// TIA Portal project "canopen-snap7-interface" (V19)
// Using a S7-1200 PLC with the CM CANopen module to interact with a CANopen and Profinet network.

(* hardware
DEVICE "S7-1200 station_1"  S7-1200 Station
   slot 0: "Rack_0"  S7-1200 Rack  Rack  V1.0
   slot 1: "PLC_1"  CPU 1215C DC/DC/DC  6ES7 215-1AG40-0XB0  V4.6
   slot 101: "CM CANopen_1"  021620-B  V1.0
*)

// ===== PLC "PLC_1"  CPU 1215C DC/DC/DC =====

VAR_GLOBAL   // PLC tag table "Standard-Variablentabelle"
   "canOpenInputs" AT %I0.0 : "typeCanProcessImageInputs";
   "canOpenOutputs" AT %Q0.0 : "typeCanProcessImageOutputs";
   "Tag_1" AT %M110.0 : Bool;
   "Tag_2" AT %M110.1 : Bool;
END_VAR

VAR_GLOBAL CONSTANT   // PLC tag table "Standard-Variablentabelle"
   "Keiner" : Pip := 65535;
   "Automatische Aktualisierung" : Pip := 0;
   "TPA 1" : Pip := 1;
   "TPA 2" : Pip := 2;
   "TPA 3" : Pip := 3;
   "TPA 4" : Pip := 4;
   "TPA OB Servo" : Pip := 32768;
   "Local~HSC_1(1)" : Hw_Hsc := 257;
   "Local~HSC_2(1)" : Hw_Hsc := 258;
   "Local~HSC_3(1)" : Hw_Hsc := 259;
   "Local~HSC_4(1)" : Hw_Hsc := 260;
   "Local~HSC_5(1)" : Hw_Hsc := 261;
   "Local~HSC_6(1)" : Hw_Hsc := 262;
   "Local~AI_2_1" : Hw_SubModule := 263;
   "Local~DI_14_DQ_10_1(1)" : Hw_SubModule := 264;
   "Local~Pulse_1(1)" : Hw_Pwm := 265;
   "Local~Pulse_2(1)" : Hw_Pwm := 266;
   "Local~Pulse_3(1)" : Hw_Pwm := 267;
   "Local~Pulse_4(1)" : Hw_Pwm := 268;
   "Local~CM_CANopen_1(1)" : Port := 270;
   "OB_Main(1)" : OB_PCYCLE := 1;
   "Local~MC(1)" : Hw_SubModule := 51;
   "Local~Common(1)" : Hw_SubModule := 50;
   "Local~Device(1)" : Hw_Device := 32;
   "Local~Configuration(1)" : Hw_SubModule := 33;
   "Local~Exec(1)" : Hw_SubModule := 52;
   "Local(1)" : Hw_SubModule := 49;
   "Local~PROFINET-Schnittstelle_1" : Hw_Interface := 64;
   "Local~PROFINET-Schnittstelle_1~Port_1" : Hw_Interface := 65;
END_VAR

TYPE "typeCanProcessImageInputs"
VERSION : 0.1
   STRUCT
      BufferA : Struct
         SlaveDigitalInput1 : Byte;
         SlaveDigitalInput2 : Byte;
         SlaveAnalogInput1 : Int;
         SlaveAnalogInput2 : Int;
         SlaveAnalogInput3 : Int;
         SlaveAnalogInput4 : Int;
      END_STRUCT;
      BufferB : Struct
         SlaveDigitalInput1 : Byte;
         SlaveDigitalInput2 : Byte;
         SlaveAnalogInput1 : Int;
         SlaveAnalogInput2 : Int;
         SlaveAnalogInput3 : Int;
         SlaveAnalogInput4 : Int;
      END_STRUCT;
      ActiveBuffer : Byte;   // 0 = BufferA, 1 = BufferB. ActiveBuffer is the buffer the PC reads from, and the inactive buffer is the buffer the PLC updates from the input CAN process image.
   END_STRUCT;
END_TYPE

TYPE "typeCanProcessImageOutputs"
VERSION : 0.1
   STRUCT
      BufferA : Struct
         SlaveDigitalOutput1 : Byte;
         SlaveDigitalOutput2 : Byte;
         SlaveAnalogOutput1 : Int;
         SlaveAnalogOutput2 : Int;
         SlaveAnalogOutput3 : Int;
         SlaveAnalogOutput4 : Int;
         RequestID : UInt;
      END_STRUCT;
      BufferB : Struct
         SlaveDigitalOutput1 : Byte;
         SlaveDigitalOutput2 : Byte;
         SlaveAnalogOutput1 : Int;
         SlaveAnalogOutput2 : Int;
         SlaveAnalogOutput3 : Int;
         SlaveAnalogOutput4 : Int;
         RequestID : UInt;
      END_STRUCT;
      ResponseID : UInt;
      ActiveBuffer : Byte;   // 0 = BufferA, 1 = BufferB. ActiveBuffer is the buffer the PLC uses to write the output process image, and the inactive buffer is the buffer the PC writes to.
   END_STRUCT;
END_TYPE

DATA_BLOCK "MappedCanProcessImageOutputs"   // DB1
{ S7_Optimized_Access := 'FALSE' }
VERSION : 0.1
   VAR
      statCanProcessImageOutputs : "typeCanProcessImageOutputs";
   END_VAR
BEGIN
   statCanProcessImageOutputs.ActiveBuffer := 16#0;
END_DATA_BLOCK

DATA_BLOCK "ControlDB"   // DB3
{ S7_Optimized_Access := 'TRUE' }
VERSION : 0.1
   VAR
      CanProcessImageIn : Array[0..31] of Byte;
      CanProcessImageOut : Array[0..9] of Byte;
      ReadCanProcessImageBusy : Bool;
      ReadCanProcessImageError : Bool;
      ReadCanProcessImageSize : UInt;
      ReadCanProcessImageStatus : DWord;
      ReadCanProcessImageValid : Bool;
      WriteCanProcessImageBusy : Bool;
      WriteCanProcessImageError : Bool;
      WriteCanProcessImageSize : UInt;
      WriteCanProcessImageStatus : DWord;
      WriteCanProcessImageDone : Bool;
      ErrorRegisterReq : Bool;
      ErrorRegisterNode : Int;
      ErrorRegisterBusy : Bool;
      ErrorRegisterGenericError : Bool;
      ErrorRegisterCurrentError : Bool;
      ErrorRegisterVoltageError : Bool;
      ErrorRegisterTemperatureError : Bool;
      ErrorRegisterCommunicationError : Bool;
      ErrorRegisterDeviceSpecificError : Bool;
      ErrorRegisterManufacturerSpecificError : Bool;
      HeartbeatReq : Bool;
      HeartbeatNode : Int;
      HeartbeatMilliseconds : UInt;
      HeartbeatBusy : Bool;
   END_VAR
BEGIN
   CanProcessImageOut[0] := 16#F0;
END_DATA_BLOCK

DATA_BLOCK "MappedCanProcessImageInputs"   // DB9
{ S7_Optimized_Access := 'FALSE' }
VERSION : 0.1
   VAR
      statCanProcessImageInputs : "typeCanProcessImageInputs";
   END_VAR
BEGIN
   statCanProcessImageInputs.ActiveBuffer := 16#0;
END_DATA_BLOCK

// folder: InstanceDBs

DATA_BLOCK "instReadCanProcessImage"   // DB5
{ S7_Optimized_Access := 'TRUE' }
VERSION : 0.1
// stored: InstanceOfName ReadCanProcessImage
"ReadCanProcessImage"
BEGIN
END_DATA_BLOCK

DATA_BLOCK "instWriteCanProcessImage"   // DB16
{ S7_Optimized_Access := 'TRUE' }
VERSION : 0.1
// stored: InstanceOfName WriteCanProcessImage
"WriteCanProcessImage"
BEGIN
END_DATA_BLOCK

// folder: (top level)

FUNCTION_BLOCK "ReadCanProcessImage"   // FB1, SCL
{ S7_Optimized_Access := 'TRUE' }
VERSION : 0.1
   VAR_OUTPUT
      Busy : Bool;
      Error : Bool;
      Len : UInt;
      Status : DWord;
      Valid : Bool;
   END_VAR
   VAR_IN_OUT
      CanProcessImage : Array[0..31] of Byte;
   END_VAR
BEGIN
   "RDREC_DB"(REQ := true,
              ID := 269,
              INDEX := 16#90,
              MLEN := 32,
              RECORD := #CanProcessImage,
              BUSY => #Busy,
              ERROR => #Error,
              LEN => #Len,
              STATUS => #Status,
              VALID => #Valid);

   // It might be an issue that REQ is always true since it uses a rising edge
   // according to ChatGPT. I haven't noticed any issues.

   // (written by Siemens dev for application example, not sure what it's for)
   // IF #Valid = true  THEN
   //     "ControlDB".Read := false;
   // END_IF;
END_FUNCTION_BLOCK

FUNCTION_BLOCK "WriteCanProcessImage"   // FB2, SCL
{ S7_Optimized_Access := 'TRUE' }
VERSION : 0.1
   VAR_OUTPUT
      Busy : Bool;
      Error : Bool;
      Status : DWord;
      Done : Bool;
   END_VAR
   VAR_IN_OUT
      CanProcessImageOutArray : Array[0..9] of Byte;
   END_VAR
BEGIN

       "WRREC_DB"(REQ := true,
                  ID := 269,
                  INDEX := 16#91,
                  LEN := 10,
                  DONE => #Done,
                  BUSY => #Busy,
                  ERROR => #Error,
                  STATUS => #Status,
                  RECORD := #CanProcessImageOutArray);

   // Changed len from 4 to 10 since my output process image is larger now. Also changed the InOut variable's array size

   // IF #Done = true  THEN
   //     "ControlDB".Write := false;
   // END_IF;
END_FUNCTION_BLOCK

FUNCTION "MapCanProcessImageToDB" : Void   // FC1, SCL
{ S7_Optimized_Access := 'TRUE' }
VERSION : 0.1
   VAR_INPUT
      ProcessImageByteArray : Array[0..31] of Byte;
   END_VAR
   VAR_IN_OUT
      CanProcessImageIn : "typeCanProcessImageInputs";
   END_VAR
BEGIN
   // Double buffer functionality implemented for asynchronous access (snap7)
   IF #CanProcessImageIn.ActiveBuffer = 0 THEN
       //map bytes 
       #CanProcessImageIn.BufferB.SlaveDigitalInput1 := #ProcessImageByteArray[0];
       #CanProcessImageIn.BufferB.SlaveDigitalInput2 := #ProcessImageByteArray[1];

       //map words
       #CanProcessImageIn.BufferB.SlaveAnalogInput1 := "BytesToWord"(Byte0 := #ProcessImageByteArray[2], Byte1 := #ProcessImageByteArray[3]);
       #CanProcessImageIn.BufferB.SlaveAnalogInput2 := "BytesToWord"(Byte0 := #ProcessImageByteArray[4], Byte1 := #ProcessImageByteArray[5]);
       #CanProcessImageIn.BufferB.SlaveAnalogInput3 := "BytesToWord"(Byte0 := #ProcessImageByteArray[6], Byte1 := #ProcessImageByteArray[7]);
       #CanProcessImageIn.BufferB.SlaveAnalogInput4 := "BytesToWord"(Byte0 := #ProcessImageByteArray[8], Byte1 := #ProcessImageByteArray[9]);

       #CanProcessImageIn.ActiveBuffer := 1;
   ELSE
       //map bytes 
       #CanProcessImageIn.BufferA.SlaveDigitalInput1 := #ProcessImageByteArray[0];
       #CanProcessImageIn.BufferA.SlaveDigitalInput2 := #ProcessImageByteArray[1];

       //map words
       #CanProcessImageIn.BufferA.SlaveAnalogInput1 := "BytesToWord"(Byte0 := #ProcessImageByteArray[2], Byte1 := #ProcessImageByteArray[3]);
       #CanProcessImageIn.BufferA.SlaveAnalogInput2 := "BytesToWord"(Byte0 := #ProcessImageByteArray[4], Byte1 := #ProcessImageByteArray[5]);
       #CanProcessImageIn.BufferA.SlaveAnalogInput3 := "BytesToWord"(Byte0 := #ProcessImageByteArray[6], Byte1 := #ProcessImageByteArray[7]);
       #CanProcessImageIn.BufferA.SlaveAnalogInput4 := "BytesToWord"(Byte0 := #ProcessImageByteArray[8], Byte1 := #ProcessImageByteArray[9]);

       #CanProcessImageIn.ActiveBuffer := 0;
   END_IF;


   //map dwords
   // Byte order reversed in application example. Not sure why as the expected byte order worked fine for me; change order as needed.

   // There aren't any dwords in use in the current program, but here is an example if needed in the future:
   // #CanProcessImageIn.SensorInPvTemperature := "BytesToDoubleWord"(Byte0 :=#ProcessImageByteArray[11],
   //                  Byte1 :=#ProcessImageByteArray[10],
   //                  Byte2 :=#ProcessImageByteArray[9],
   //                  Byte3 :=#ProcessImageByteArray[8]);
   //                  

   // To avoid using functions for this process, use slice notation:
   //     #CanProcessImageIn.SlaveAnalogInput1.%B0 := #ProcessImageByteArray[3]; // Low byte
   //     #CanProcessImageIn.SlaveAnalogInput1.%B1 := #ProcessImageByteArray[2]; // High byte
END_FUNCTION

FUNCTION "BytesToWord" : Word   // FC2, SCL
{ S7_Optimized_Access := 'TRUE' }
VERSION : 0.1
   VAR_INPUT
      Byte0 : Byte;
      Byte1 : Byte;
   END_VAR
BEGIN
   //This block turns two bytes into a word (little-endian)
   //The order of bytes within the resulting word is: B1B0

   //Example: Byte0 is 1111111 and Byte1 is 10101010
   //This operation will add Byte0 (1111111) to the 8-bit-leftshifted version of Byte1 (10101010 00000000)
   //10101010 00000000 + 11111111
   //Result Word = 10101010 11111111
   #BytesToWord := BYTE_TO_WORD(IN:=#Byte0) + SHL(IN := BYTE_TO_WORD(IN:=#Byte1), N := 8);
END_FUNCTION

FUNCTION "BytesToDoubleWord" : DWord   // FC3, SCL
{ S7_Optimized_Access := 'TRUE' }
VERSION : 0.1
   VAR_INPUT
      Byte0 : Byte;
      Byte1 : Byte;
      Byte2 : Byte;
      Byte3 : Byte;
   END_VAR
   VAR_TEMP
      tempWord0 : Word;
      tempWord1 : Word;
   END_VAR
BEGIN
   //This function block creates a Dword out of four bytes
   //The order of bytes within the resulting Dword is: B3B2B1B0


   #tempWord0:= "BytesToWord"(Byte0 := #Byte0, Byte1 := #Byte1);
   #tempWord1 := "BytesToWord"(Byte0 := #Byte2, Byte1 := #Byte3);

   #BytesToDoubleWord := WORD_TO_DWORD(IN:=#tempWord0) + SHL(IN := WORD_TO_DWORD(IN:=#tempWord1), N := 16);
END_FUNCTION

FUNCTION "InvertWordEndianness" : Word   // FC5, SCL
{ S7_Optimized_Access := 'FALSE' }
VERSION : 0.1
   VAR_INPUT
      InputWord : Word;
   END_VAR
   VAR_TEMP
      tempInputByte0 : Byte;
      tempInputByte1 : Byte;
   END_VAR
BEGIN
   #tempInputByte0 := WORD_TO_BYTE(#InputWord & 2#0000000011111111); // Least significant portion of word (little-endian)
   #tempInputByte1 := WORD_TO_BYTE(SHR(IN:=#InputWord, N:=8));       // Most significant portion of word (little-endian)  

   // I believe this code is incorrect. #tempInputByte0 and #tempInputByte1 should be swapped to invert the endianness
   #InvertWordEndianness := "BytesToWord"(Byte0 := #tempInputByte0, Byte1 := #tempInputByte1);
END_FUNCTION

FUNCTION "WordToBytes" : Void   // FC6, SCL
{ S7_Optimized_Access := 'TRUE' }
VERSION : 0.1
   VAR_INPUT
      "Word" : Word;
   END_VAR
   VAR_OUTPUT
      Byte0 : Byte;
      Byte1 : Byte;
   END_VAR
BEGIN
   #Byte0 := WORD_TO_BYTE(#Word AND 2#0000000011111111);
   #Byte1 := WORD_TO_BYTE(SHR(IN := #Word, N := 8));
END_FUNCTION

FUNCTION "MapDBToCanProcessImage" : Void   // FC7, SCL
{ S7_Optimized_Access := 'TRUE' }
VERSION : 0.1
   VAR_OUTPUT
      ProcessImageByteArray : Array[0..9] of Byte;
   END_VAR
   VAR_IN_OUT
      CanProcessImageOut : "typeCanProcessImageOutputs";
   END_VAR
BEGIN
   // Double buffer functionality and handshake implemented for asynchronous access (snap7)
   IF #CanProcessImageOut.ActiveBuffer = 0 THEN
       // map bytes
       #ProcessImageByteArray[0] := #CanProcessImageOut.BufferA.SlaveDigitalOutput1;
       #ProcessImageByteArray[1] := #CanProcessImageOut.BufferA.SlaveDigitalOutput2;

       //map words
       "WordToBytes"("Word" := #CanProcessImageOut.BufferA.SlaveAnalogOutput1,
                     Byte0 => #ProcessImageByteArray[2],
                     Byte1 => #ProcessImageByteArray[3]);
       "WordToBytes"("Word" := #CanProcessImageOut.BufferA.SlaveAnalogOutput2,
                     Byte0 => #ProcessImageByteArray[4],
                     Byte1 => #ProcessImageByteArray[5]);
       "WordToBytes"("Word" := #CanProcessImageOut.BufferA.SlaveAnalogOutput3,
                     Byte0 => #ProcessImageByteArray[6],
                     Byte1 => #ProcessImageByteArray[7]);
       "WordToBytes"("Word" := #CanProcessImageOut.BufferA.SlaveAnalogOutput4,
                     Byte0 => #ProcessImageByteArray[8],
                     Byte1 => #ProcessImageByteArray[9]);

       #CanProcessImageOut.ResponseID := #CanProcessImageOut.BufferA.RequestID;
   ELSE
       // map bytes
       #ProcessImageByteArray[0] := #CanProcessImageOut.BufferB.SlaveDigitalOutput1;
       #ProcessImageByteArray[1] := #CanProcessImageOut.BufferB.SlaveDigitalOutput2;

       //map words
       "WordToBytes"("Word" := #CanProcessImageOut.BufferB.SlaveAnalogOutput1,
                     Byte0 => #ProcessImageByteArray[2],
                     Byte1 => #ProcessImageByteArray[3]);
       "WordToBytes"("Word" := #CanProcessImageOut.BufferB.SlaveAnalogOutput2,
                     Byte0 => #ProcessImageByteArray[4],
                     Byte1 => #ProcessImageByteArray[5]);
       "WordToBytes"("Word" := #CanProcessImageOut.BufferB.SlaveAnalogOutput3,
                     Byte0 => #ProcessImageByteArray[6],
                     Byte1 => #ProcessImageByteArray[7]);
       "WordToBytes"("Word" := #CanProcessImageOut.BufferB.SlaveAnalogOutput4,
                     Byte0 => #ProcessImageByteArray[8],
                     Byte1 => #ProcessImageByteArray[9]);

       #CanProcessImageOut.ResponseID := #CanProcessImageOut.BufferB.RequestID;
   END_IF;


   // The byte order for the WordToBytes calls were originally swapped in the application example, so I left
   // this comment, but it is not true for this program (not sure why):
   // Byte order is swapped since the CanProcessImageOut DB is non-optimized (big-endian) and everything else uses little-endian
END_FUNCTION

ORGANIZATION_BLOCK "Main"   // OB1, LAD, ProgramCycle
TITLE = "Main Program Sweep (Cycle)"
{ S7_Optimized_Access := 'TRUE' }
VERSION : 0.1
   VAR_INPUT
      Initial_Call : Bool;   // Initial call of this OB
      Remanence : Bool;   // =True, if remanent data are available
   END_VAR
BEGIN

REGION Network 1
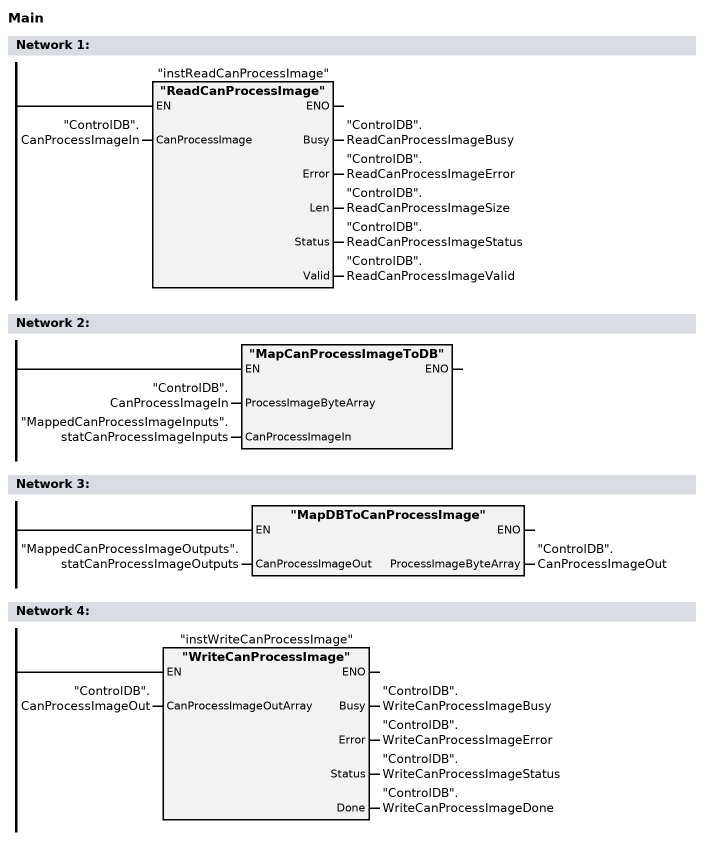
   RUNG wire#powerrail
      "instReadCanProcessImage"(CanProcessImage := "ControlDB".CanProcessImageIn, Busy => "ControlDB".ReadCanProcessImageBusy, Error => "ControlDB".ReadCanProcessImageError, Len => "ControlDB".ReadCanProcessImageSize, Status => "ControlDB".ReadCanProcessImageStatus, Valid => "ControlDB".ReadCanProcessImageValid)
   END_RUNG
   // the same network as SCL:
   "instReadCanProcessImage"(CanProcessImage := "ControlDB".CanProcessImageIn,   // "ReadCanProcessImage"
                           Busy => "ControlDB".ReadCanProcessImageBusy,
                           Error => "ControlDB".ReadCanProcessImageError,
                           Len => "ControlDB".ReadCanProcessImageSize,
                           Status => "ControlDB".ReadCanProcessImageStatus,
                           Valid => "ControlDB".ReadCanProcessImageValid);
END_REGION

REGION Network 2
   RUNG wire#powerrail
      "MapCanProcessImageToDB"(ProcessImageByteArray := "ControlDB".CanProcessImageIn, CanProcessImageIn := "MappedCanProcessImageInputs".statCanProcessImageInputs)
   END_RUNG
   // the same network as SCL:
   "MapCanProcessImageToDB"(ProcessImageByteArray := "ControlDB".CanProcessImageIn,
                           CanProcessImageIn := "MappedCanProcessImageInputs".statCanProcessImageInputs);
END_REGION

REGION Network 3
   RUNG wire#powerrail
      "MapDBToCanProcessImage"(CanProcessImageOut := "MappedCanProcessImageOutputs".statCanProcessImageOutputs, ProcessImageByteArray => "ControlDB".CanProcessImageOut)
   END_RUNG
   // the same network as SCL:
   "MapDBToCanProcessImage"(CanProcessImageOut := "MappedCanProcessImageOutputs".statCanProcessImageOutputs,
                           ProcessImageByteArray => "ControlDB".CanProcessImageOut);
END_REGION

REGION Network 4
   RUNG wire#powerrail
      "instWriteCanProcessImage"(CanProcessImageOutArray := "ControlDB".CanProcessImageOut, Busy => "ControlDB".WriteCanProcessImageBusy, Error => "ControlDB".WriteCanProcessImageError, Status => "ControlDB".WriteCanProcessImageStatus, Done => "ControlDB".WriteCanProcessImageDone)
   END_RUNG
   // the same network as SCL:
   "instWriteCanProcessImage"(CanProcessImageOutArray := "ControlDB".CanProcessImageOut,   // "WriteCanProcessImage"
                           Busy => "ControlDB".WriteCanProcessImageBusy,
                           Error => "ControlDB".WriteCanProcessImageError,
                           Status => "ControlDB".WriteCanProcessImageStatus,
                           Done => "ControlDB".WriteCanProcessImageDone);
END_REGION
END_ORGANIZATION_BLOCK